FUNCTION_BLOCK DIAG_LOG (* A diagnostic log with time stamping of conditions,acknowledgments and repair times *)
  (* Standard: 61499-1; Classification: HMI; ApplicationDomain: Diagnostics; Function: Tabular log *)
  (* Version 0.1, 2004-06-23, JHC, Rockwell Automation, Moved to fb.rt.swing, subclassed from FB_TABLE. *)
  (* Version 0.0, 2001-04-14, JHC, Rockwell Automation, First XML version *)
  (* Compiler header: package fb.rt.swing; *)
  (* Compiler classdef: public class DIAG_LOG extends FB_TABLE *)
  (* Compiler Java Sun JDK 1.4.2 *)
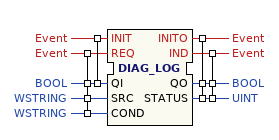
  EVENT_INPUT
    INIT WITH QI; (* Initialize *)
    REQ WITH SRC, COND, QI; (* Log an event *)
  END_EVENT
  EVENT_OUTPUT
    INITO WITH STATUS, QO; (* Initialization Confirm *)
    IND WITH QO, STATUS; (* REQ Confirmation *)
  END_EVENT
  VAR_INPUT
    QI : BOOL; (* Input event qualifier (see FB_TABLE for usage) *)
    SRC : WSTRING; (* Source of event being logged *)
    COND : WSTRING; (* Condition being logged *)
  END_VAR
  VAR_OUTPUT
    QO : BOOL; (* Output qualifier, (see FB_TABLE for usage) *)
    STATUS : UINT; (* 0=OK,2=TYPE_CONVERSION_ERROR,4=INHIBITED,13=ARRAY_SIZE_ERROR *)
  END_VAR
END_FUNCTION_BLOCK
